// TwinCAT 3 PLC project Damper
// ProgramVersion: 3.1.4024.0
// libraries:
//   Tc2_HVAC, * (Beckhoff Automation GmbH)
//   Tc2_MC2, * (Beckhoff Automation GmbH)
//   Tc2_Standard, * (Beckhoff Automation GmbH)
//   Tc2_System, * (Beckhoff Automation GmbH)
//   Tc3_Module, * (Beckhoff Automation GmbH)
//   VisuSymbols,3.5.10.0,System
// project tree:
//   / GlobalTextList.TcGTLO, PlcTask.TcTTO, SensorTask.TcTTO, Visualization Manager.TcVMO (not stored)
//   POUs/ FB_ReadAccelerometer.TcPOU (not stored), MAIN.TcPOU (not stored), P_ReadSesnors.TcPOU
//   VISUs/ Visualization.TcVIS (not stored)
// real-time tasks:
//   TASK PlcTask: cycle T#10ms, priority 10, ADS port 350
//   TASK TcCOM Task: cycle T#5ms, priority 20, ADS port 351
//   TASK SensorTask: cycle T#10ms, priority 30, ADS port 352
// motion (NC):
//   TASK NC-Task 1 SAF: cycle T#2ms, priority 4, ADS port 501
//   TASK NC-Task 1 SVB: cycle T#10ms, priority 8, ADS port 511
//   AXIS Drive (id 1)
//     Dynamic: AccelerationMaximum=1500, DecelerationMaximum=5000, Acceleration=1000, Deceleration=333
//     Velo: Maximum=1000
//     PositionAreaControl: Enable=false
//     TargetPosControl: Enable=false
//     OtherSettings: AllowMotionCmdToSlave=true
//     encoder EncType=19
//       EncPara: ScaleFactorNumerator=0.02275, ModuloFactor=187, MaxCount=#xffffffff
//         SoftEndMinControl: Range=2
//         SoftEndMaxControl: Range=185
//     drive DrvType=16
//       DrvPara: MaxCount=#xffffffff
//         Analog: VeloReferenz=1000, TorqueSetpointScale=10, ScaleFactorActTorque=0.1
//         TimeComp: TaskDelayCycles=1
//     controller CtrType=1
//       CtrPara: PriorControlFactor=1
//         PosDiffControl: Enable=false
//         Observer: BandWidth=20
// I/O:
//   DEVICE EtherCAT Port, AmsNetId 134.28.120.143.4.1
//     EtherCAT Terminal (EK1100) [EK1100 EtherCAT Coupler (2A E-Bus)]
//       Digital Terminal (EL1814) [EL1814 4Ch. Dig. Input 24V, 10µs]
//       Accelerometer Terminal (ELM3604-0002) [ELM3604-0002 4Ch. IEPE Sensor, 24 bit, high precision]
//       End Cap (EL9011) [EL9011 End Terminal]
//     Drive (MC3603) [MC3603 MotionController]
// variable links:
//   EtherCAT Port <-> TcCOM Objects/Damper
//     Drive (MC3603)/Receive PDO4 mapping / Number of mapped objects/Target torque <-> damper_twincat_Y/torque
//   NC-Task 1 SAF/Axes/Drive <-> EtherCAT Port/Drive (MC3603)
//     Drive/Inputs/In/nDataIn3[0] <-> Transmit PDO4 mapping  / Number of mapped objects/Torque actual value
//     Drive/Inputs/In/nDcOutputTime <-> InfoData/DcOutputShift
//     Drive/Inputs/In/nState1 <-> Transmit PDO4 mapping  / Number of mapped objects/Statusword
//     Drive/Inputs/In/nState2 <-> Transmit PDO4 mapping  / Number of mapped objects/Statusword @bit 8
//     Drive/Inputs/In/nState4 @bit 1 <-> WcState/InputToggle
//     Drive/Inputs/In/nState4 <-> WcState/WcState
//     Drive/Outputs/Out/nCtrl1 <-> Receive PDO4 mapping / Number of mapped objects/Controlword
//     Drive/Outputs/Out/nCtrl2 <-> Receive PDO4 mapping / Number of mapped objects/Controlword @bit 8
//   Damper/Damper Instance <-> EtherCAT Port/Drive (MC3603)
//     SensorTask Outputs/MAIN.iTorqueOffset <-> Receive PDO4 mapping / Number of mapped objects/Torque offset
//   Damper/Damper Instance <-> EtherCAT Port/EtherCAT Terminal (EK1100)/Accelerometer Terminal (ELM3604-0002)
//     SensorTask Inputs/P_ReadSesnors.fbReadAcc.c1Sample <-> PAI Samples 1 Channel 1/Samples[0]
//     SensorTask Inputs/P_ReadSesnors.fbReadAcc.c2Sample <-> PAI Samples 1 Channel 2/Samples[0]
//     SensorTask Inputs/P_ReadSesnors.fbReadAcc.c3Sample <-> PAI Samples 1 Channel 3/Samples[0]
//   Damper/Damper Instance <-> NC-Task 1 SAF/Axes/Drive
//     PlcTask Inputs/MAIN.drive.NcToPlc <-> Outputs/ToPlc
//     PlcTask Outputs/MAIN.drive.PlcToNc <-> Inputs/FromPlc
//   Damper/Damper Instance <-> TcCOM Objects/Damper
//     PlcTask Outputs/MAIN.bRun <-> damper_twincat_U/enable
//     SensorTask Outputs/P_ReadSesnors.accZ <-> damper_twincat_U/acc

CONFIGURATION Damper
    RESOURCE PLC ON TwinCAT3
        TASK PlcTask(INTERVAL := T#10ms, PRIORITY := 10);
        TASK SensorTask(INTERVAL := T#10ms, PRIORITY := 30);
        PROGRAM MAIN WITH PlcTask : MAIN;
        PROGRAM P_ReadSesnors WITH SensorTask : P_ReadSesnors;
    END_RESOURCE
END_CONFIGURATION

// ---- POUs/P_ReadSesnors.TcPOU
PROGRAM P_ReadSesnors
VAR
	fbReadAcc : FB_ReadAccelerometer;
	
	accX AT %Q* : LREAL;
	accY AT %Q* : LREAL;
	accZ AT %Q* : LREAL;
END_VAR

fbReadAcc(accX=>accX, accY=>accY, accZ=>accZ);

END_PROGRAM
